PROGRAM Analogue_Processing
VAR
END_VAR

Temperature_Transducer_A1(RawValue	:=	Temperature_Transducer_A1_Raw_Value);

END_PROGRAM

(* stored: Version 1.1.0.1, ProductVersion 3.1.4024.15
   POU Analogue_Processing: Id {d9437fd0-b491-47b7-8255-0da34a1bfe69}, SpecialFunc None *)
